// TwinCAT 3 PLC project Unbenannt2
// ProgramVersion: 3.1.0.9
// libraries:
//   Standard, * (System)
//   Tc2_Standard, * (Beckhoff Automation GmbH)
//   Tc2_System, * (Beckhoff Automation GmbH)
//   Tc3_Interfaces, * (Beckhoff Automation GmbH)
//   Tc3_Module, * (Beckhoff Automation GmbH)
// project tree:
//   / PlcTask.TcTTO
//   POUs/ Converter.TcPOU, MAIN.TcPOU, Ob.TcPOU, Ob2.TcPOU
// real-time tasks:
//   TASK PlcTask: cycle T#10ms, priority 20, ADS port 350
//   TASK Task 3: cycle T#10ms, priority 1, ADS port 351
// variable links:
//   Unbenannt2/Unbenannt2 Instance <-> TcCOM Objects/Object2 (CModule1)
//     PlcTask Inputs/MAIN.In <-> Outputs/Value
//     PlcTask Outputs/MAIN.Out <-> Inputs/Value
//     PlcTask Outputs/MAIN.Reset <-> Inputs/Rst
//   Unbenannt2/Unbenannt2 Instance <-> TcCOM Objects/Object3 (CModule1)
//     PlcTask Outputs/MAIN.Out <-> Inputs/Value

CONFIGURATION Unbenannt2
    RESOURCE PLC ON TwinCAT3
        TASK PlcTask(INTERVAL := T#10ms, PRIORITY := 20);
        PROGRAM MAIN WITH PlcTask : MAIN;
    END_RESOURCE
END_CONFIGURATION

// ---- POUs/MAIN.TcPOU
PROGRAM MAIN
VAR
	In AT %I* : UDINT;
	Out AT %Q* : UDINT;
	Reset AT %Q* : BOOL;
	Intern1 : UDINT;
	Intern2 : UDINT;
	Intern3 : UDINT;
	Obj1 : Ob2;
	Obj2 : Ob2;
END_VAR

IF In < 800
	THEN 	Out := 5;
			Reset := FALSE;
ELSIF In < 1000
	THEN 	Out := 2;
ELSE
	Out := 0;
	Reset := TRUE;
	Ob.Doub();
	Obj1.DefL(Intern3);
	Obj2.DefL(Intern2);
END_IF

Intern3 := Converter(Intern1,Intern2);

Intern1 := Ob.Val();
Intern2 := Obj1.Area();
Obj2.Area();

END_PROGRAM

// ---- POUs/Ob2.TcPOU
FUNCTION_BLOCK Ob2
VAR_INPUT
END_VAR
VAR_OUTPUT
END_VAR
VAR
	Length : UDINT := 3;
	Height : UDINT := 2;
END_VAR

METHOD Area : UDINT
VAR_INPUT
END_VAR
Area := Length * Height;
END_METHOD

METHOD DefL : UDINT
VAR_INPUT
	L : UDINT;
END_VAR
Length := L;
DefL := Length;
END_METHOD

END_FUNCTION_BLOCK

// ---- POUs/Ob.TcPOU
PROGRAM Ob
VAR
	In1 : UDINT;
END_VAR

ACTION Doub:
In1 := 2*In1;
END_ACTION

METHOD FB_init : BOOL
VAR_INPUT
	bInitRetains : BOOL; // if TRUE, the retain variables are initialized (warm start / cold start)
	bInCopyCode : BOOL;  // if TRUE, the instance afterwards gets moved into the copy code (online change)
END_VAR
In1 := 5;
END_METHOD

METHOD Load : UDINT
VAR_INPUT
	Input : UDINT;
END_VAR
In1 := Input;
Load := In1;
END_METHOD

METHOD Val : UDINT
VAR_INPUT
END_VAR
Val := In1;
END_METHOD

END_PROGRAM

// ---- POUs/Converter.TcPOU
FUNCTION Converter : UDINT
VAR_INPUT
	CIn1 : UDINT;
	CIn2 : UDINT;
END_VAR
VAR
	Intern3 : UDINT;
END_VAR

Intern3 := CIn1 + CIn2;
Converter := Intern3;

END_FUNCTION
